TYPE ST_NeedleAllocatefeeback :
STRUCT
	//領取盒子的狀態
	BoxStatus		:		E_BoxStatus;
	//所需盒數
	Box				:       INT;
END_STRUCT
END_TYPE

(* stored: Version 1.1.0.1, ProductVersion 3.1.4024.13
   DUT ST_NeedleAllocatefeeback: Id {875b1b5b-a4a1-4bb8-b82c-80b1f8ae10f2} *)
